FUNCTION_BLOCK OGD251_Decoder IMPLEMENTS I_DisSensor
VAR_INPUT
	// 關閉感應器
	DisableSeosor :	BOOL;
END_VAR
VAR_OUTPUT
	// 距離 (單位:mm)
	fDistance : REAL;
	// 裝置狀態正常
	SSC1_1			:BOOL;
	// 裝置狀態正常
	bDevice_is_OK			:BOOL;
	// 需要維護
	bMaintenance_required	:BOOL;
	// 超出測量距離
	bOut_of_specification	:BOOL;
	// 檢查功能
	bFunctional_check		:BOOL;
	// 錯誤
	bFailure				:BOOL;
	// 距離比例(單位:公尺)
	iScale_Distance			:INT;
END_VAR
VAR
	// 原始資料輸入
	in_RawData AT %I* : ARRAY [0..7] OF USINT;
	// 原始資料輸出
	out_rawdata AT %Q* :USINT;	
	
	

	DistanceTmp : WORD;
	tmpStatus : WORD;
	tmpStatus2 : WORD;
	tmpStatus3 : POINTER TO SINT;
	tmpfDistance : SINT;
END_VAR

DistanceTmp := USINT_TO_WORD(in_RawData[0]);

DistanceTmp := ROL(DistanceTmp, 8) + USINT_TO_WORD(in_RawData[1]);


// 數值比例 (單位:公尺)
tmpStatus3 := ADR(in_RawData[2]);




IF (DistanceTmp = 16#7FF8) OR (DistanceTmp = 16#8008) OR (DistanceTmp = 16#7FFC) THEN
	fDistance := 0;
ELSE
	// 距離 = 感應器RAW值 X 10^單位值 X 1000(將 m 轉為 mm)
	fDistance := LREAL_TO_REAL(DistanceTmp * EXPT(10, tmpStatus3^) * 1000);
END_IF

tmpStatus := ROR(in_RawData[3] AND 16#F0, 4);

SSC1_1 := (in_RawData[3] AND 16#1) = 1;

bDevice_is_OK := tmpStatus = 0;
bMaintenance_required := tmpStatus = 1;
bOut_of_specification := tmpStatus = 2;
bFunctional_check := tmpStatus = 3;
bFailure := tmpStatus = 4;

tmpStatus2 := 0;
tmpStatus2.0 := DisableSeosor;

out_rawdata := WORD_TO_USINT(tmpStatus2);

PROPERTY Distance : REAL
GET
Distance := fDistance;
END_GET
END_PROPERTY

END_FUNCTION_BLOCK

(* stored: Version 1.1.0.1, ProductVersion 3.1.4024.15
   POU OGD251_Decoder: Id {91d286db-3331-48bf-a248-2311590c3f23}, SpecialFunc None
   Property Distance: Id {8e0378c0-67bb-40cd-9e30-84522ca06113}
   Get Get: Id {e7885e92-8d61-48f1-bb65-3b7427544fc6} *)
